// TIA Portal project "Project1" (V20)

(* hardware
DEVICE "S7-1500/ET200MP station_1"  S7-1500 station
   slot 0: "Rail_0"  Rack  6ES7 590-1***0-0AA0
   slot 1: "PLC_1"  CPU 1516F-3 PN/DP  6ES7 516-3FN00-0AB0  V1.8
      slot 3: "CPU display_1"  6ES7591-1BA00-0AA0
      slot 32768: "PROFINET interface_1"  X1
         slot 32769: "Port_1"  X1 P1
         slot 32770: "Port_2"  X1 P2
      slot 33024: "PROFINET interface_2"  X2
         slot 33025: "Port_1"  X2 P1
      slot 33280: "DP interface_1"  X3
   slot 2: "F-DI 16x24V DC_1"  F-DI 16x24V DC  6ES7 526-1BH00-0AB0  V1.0
      slot 1: "F-DI 16x24V DC_1"  F-DI 16x24V DC
   slot 3: "F-DQ 8x24V DC/2A PPM_1"  F-DQ 8x24V DC/2A PPM  6ES7 526-2BF00-0AB0  V1.0
      slot 1: "F-DQ 8x24V DC/2A PPM_1"  F-DQ 8x24V DC/2A PPM
   slot 4: "DI 16x24VDC BA_1"  DI 16x24VDC BA  6ES7 521-1BH10-0AA0  V1.1
*)

// ===== PLC "PLC_1"  CPU 1516F-3 PN/DP =====
// protected blocks, not shown: "Main_Safety_RTG1", "Main_Safety_RTG1_DB"

VAR_GLOBAL   // PLC tag table "Default tag table"
   "E-Stop" AT %I0.0 : Bool;
   "Motor" AT %Q9.0 : Bool;
   "Acknowledge" AT %I15.0 : Bool;
   "PF_OSSD" AT %I0.1 : Bool;
   "WF_Clear" AT %I0.2 : Bool;
   "ENC_A" AT %IW100 : Int;
   "ENC_B" AT %IW102 : Int;
   "CASE_B0" AT %Q9.1 : Bool;
   "CASE_B1" AT %Q9.2 : Bool;
   "V_Limit" AT %MW100 : Int;
   "PF_OSSD_right" AT %I0.3 : Bool;
   "WF_Clear_right" AT %I0.4 : Bool;
   "PF_OSSD_left" AT %I0.5 : Bool;
   "WF_Clear_left" AT %I0.6 : Bool;
END_VAR

ORGANIZATION_BLOCK "Main"   // OB1, FBD, ProgramCycle
TITLE = "Main Program Sweep (Cycle)"
{ S7_Optimized_Access := 'TRUE' }
VERSION : 0.1
   VAR_INPUT
      Initial_Call : Bool;   // Initial call of this OB
      Remanence : Bool;   // =True, if remanent data are available
   END_VAR
   VAR_TEMP
      wf : Bool;
   END_VAR
BEGIN

REGION Network 1
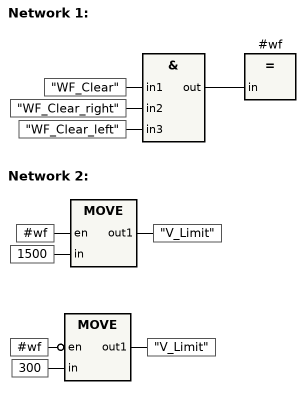
   #wf := "WF_Clear" AND "WF_Clear_right" AND "WF_Clear_left";
END_REGION

REGION Network 2
   IF #wf THEN "V_Limit" := 1500; END_IF;
   IF NOT #wf THEN "V_Limit" := 300; END_IF;
END_REGION
END_ORGANIZATION_BLOCK